ABB RobotStudio station: Solution38RISA.rspag

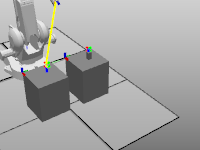
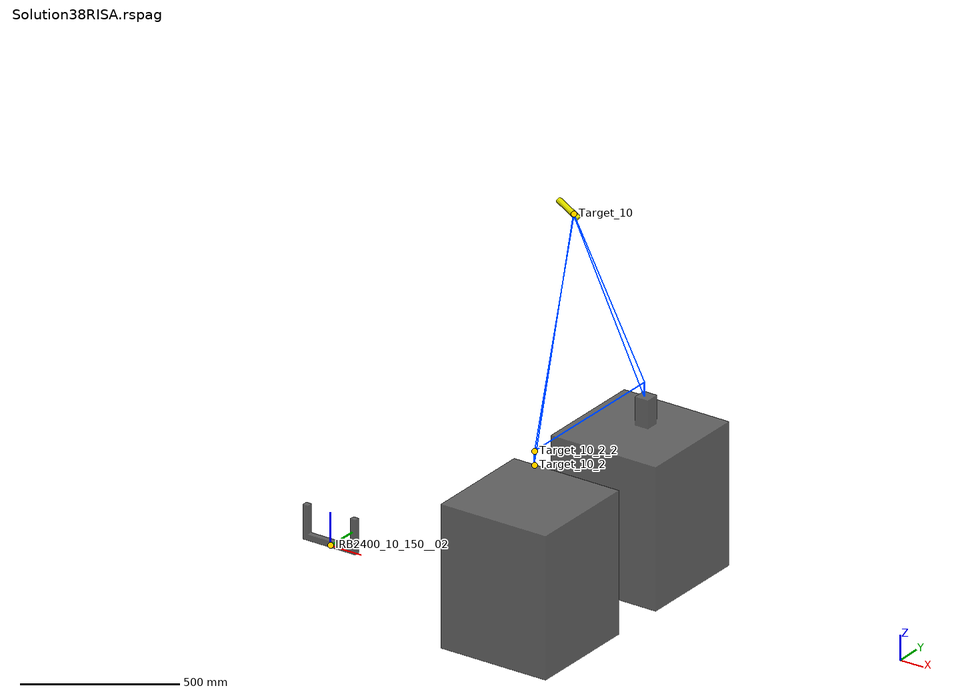
[picture v1: parts stored in the station drawn from their meshes, with robot base, taught points and paths (robot models come from the ABB library and are not in the file)]
--- station ---
Station Solution38RISA (saved by RobotStudio 21.4.9700.0)
Controller IRB2400_10_150
  mechanical unit ROB_1: IRB2400_10_150__02, 6 joints, base frame (0, 0, 0) mm
Layout (positions relative to the parent item):
  - IRB2400_10_150__02 [mechanism, from Robots\IRB2400_10_150_G_02.rslib] at (0, 0, 0) mm; joint values [0, -0.1065, -0.072, 0, 0.5956, 0] (rad or m)
  - Part_4 [part], size 400 x 400 x 500 mm
  - Part_5 [part] at (0, 600, 0) mm, size 400 x 400 x 500 mm
  - Part_6 [part] at (75.01, 607.78, -200) mm, size 50 x 50 x 100 mm
  - Part_1 [part], size 200 x 20 x 20 mm
    - My_Tool1_1 [frame] at (0, 0, 100) mm
  - Part_2 [part], size 20 x 20 x 100 mm
  - Part_3 [part], size 20 x 20 x 100 mm
  - SCGripper1 [smart component] at (842.01, 0, 1462.5) mm, rotated rx -180 ry 60 rz -180 deg
      signals: DI SCOpen, DI SCClose, DO SCClosed, DO SCOpened, DO SCDetal
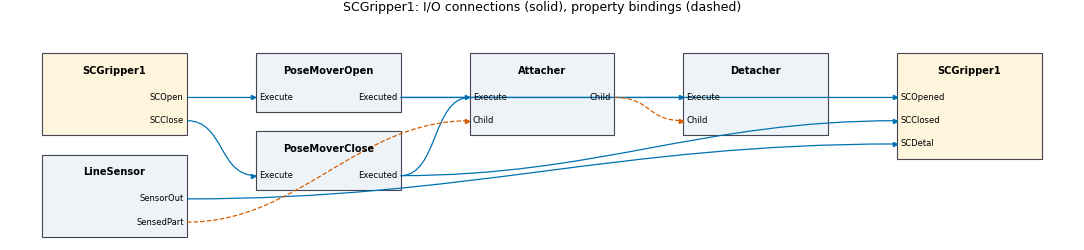
      connections:
        SCGripper1.SCOpen -> PoseMoverOpen.Execute
        SCGripper1.SCClose -> PoseMoverClose.Execute
        PoseMoverOpen.Executed -> SCGripper1.SCOpened
        PoseMoverClose.Executed -> SCGripper1.SCClosed
        LineSensor.SensorOut -> SCGripper1.SCDetal
        PoseMoverClose.Executed -> Attacher.Execute
        PoseMoverOpen.Executed -> Detacher.Execute
        LineSensor.SensedPart => Attacher.Child
        Attacher.Child => Detacher.Child
    - My_Tool1 [mechanism] at (0, 0, 0) mm; joint values [0, 0] (rad or m)
        TCP My_Tool1_1 at (0, 0, 100) mm
        links: L1, L2, L3
    - PoseMoverOpen [smart component, from Components\PoseMover.rslib]
        properties: Mechanism=My_Tool1; Pose=2; Duration=2
    - PoseMoverClose [smart component, from Components\PoseMover.rslib]
        properties: Mechanism=My_Tool1; Pose=3; Duration=2
    - LineSensor [smart component, from Components\LineSensor.rslib]
        properties: Start=[0 0 0.03]; End=[0 0 0.12]; Radius=0.01; SensedPart=(none); SensedPoint=[0 0 0]
      - _sensorPart_ [part], size 20 x 20 x 90 mm
    - Attacher [smart component, from Components\Attacher.rslib]
        properties: Parent=My_Tool1; Flange=0; Child=(none); Mount=false; Offset=[0 0 0]; Orientation=[0 0 0]
    - Detacher [smart component, from Components\Detacher.rslib]
        properties: Child=(none); KeepPosition=true
Attachment: SCGripper1 is attached to IRB2400_10_150__02 / Link6
Attachment: Workobject_1 is attached to Part_4
Attachment: Workobject_2 is attached to Part_5
Collision set CollisionSet_1: My_Tool1 against Part_6, near miss 0 m
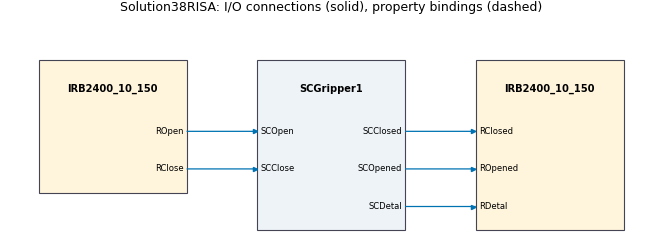
Station logic (signal -> signal, property => property):
  IRB2400_10_150.ROpen -> SCGripper1.SCOpen
  IRB2400_10_150.RClose -> SCGripper1.SCClose
  SCGripper1.SCClosed -> IRB2400_10_150.RClosed
  SCGripper1.SCOpened -> IRB2400_10_150.ROpened
  SCGripper1.SCDetal -> IRB2400_10_150.RDetal
Targets, tools, work objects and paths stored in the station and not in the controller backup, written as RAPID:
! task T_ROB1
MODULE Module1
  CONST robtarget Target_10_2_3:=[[200,225,100],[0,0,1,0],[-1,0,-1,0],[9E+09,9E+09,9E+09,9E+09,9E+09,9E+09]];
  CONST robtarget Target_10_2_2_2:=[[200,225,150],[0,0,1,0],[-1,0,1,0],[9E+09,9E+09,9E+09,9E+09,9E+09,9E+09]];
ENDMODULE


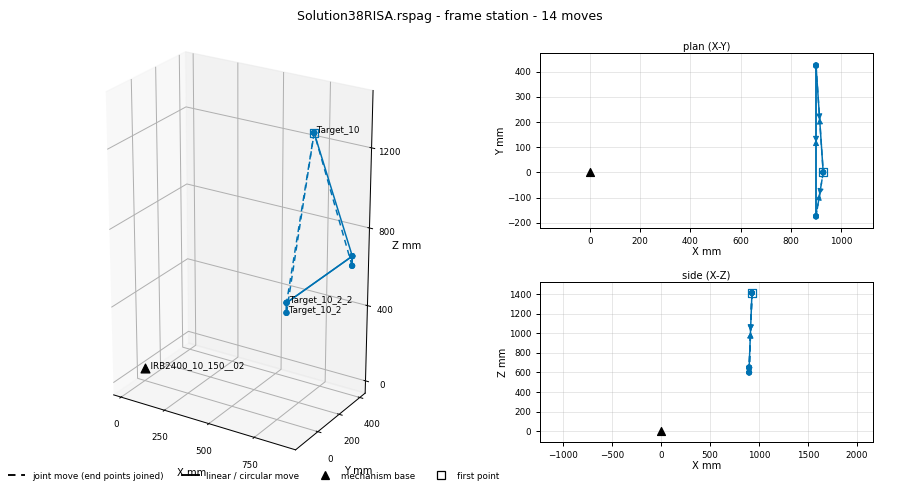
[picture p0: tool path of Solution38RISA.rspag in frame station, 14 of 14 moves have a stored position in this frame; points joined in program order, loops and branches not executed]
--- Backups/IRB2400_10_150/RAPID/TASK1/PROGMOD/CalibData.mod ---
MODULE CalibData
    TASK PERS wobjdata Workobject_1:=[FALSE,TRUE,"",[[700,-400,500],[1,0,0,0]],[[0,0,0],[1,0,0,0]]];
    TASK PERS wobjdata Workobject_2:=[FALSE,TRUE,"",[[700,200,500],[1,0,0,0]],[[0,0,0],[1,0,0,0]]];
    PERS tooldata Tooldata_1:=[TRUE,[[0,0,100],[1,0,0,0]],[1,[0,0,1],[1,0,0,0],0,0,0]];
ENDMODULE

--- Backups/IRB2400_10_150/RAPID/TASK1/PROGMOD/Module1.mod ---
MODULE Module1
        CONST robtarget Target_10:=[[928.612159322,0,1412.5],[0.5,0,0.866025404,0],[0,0,0,0],[9E+09,9E+09,9E+09,9E+09,9E+09,9E+09]];
    CONST robtarget Target_10_2_2:=[[200,225,150],[0,0,1,0],[-1,0,1,0],[9E+09,9E+09,9E+09,9E+09,9E+09,9E+09]];
    CONST robtarget Target_10_2:=[[200,225,100],[0,0,1,0],[-1,0,-1,0],[9E+09,9E+09,9E+09,9E+09,9E+09,9E+09]];
!***********************************************************
    !
    ! Module:  Module1
    !
    ! Description:
    !   <Insert description here>
    !
    ! Author: srk
    !
    ! Version: 1.0
    !
    !***********************************************************


    !***********************************************************
    !
    ! Procedure main
    !
    !   This is the entry point of your program
    !
    !***********************************************************
    PROC main()
        !Add your code here
    ENDPROC
    PROC Path_10()
        MoveJ Target_10,v1000,fine,Tooldata_1\WObj:=wobj0;
        Reset ROpen;
        Reset RClose;
        Set ROpen;
        WaitDI ROpened, 1;
        Reset ROpen;
        MoveJ Target_10_2_2,v1000,z30,Tooldata_1\WObj:=Workobject_1;
        MoveL Target_10_2,v100,fine,Tooldata_1\WObj:=Workobject_1;
        IF RDetal=1 THEN
        Set RClose;
        WaitDI RClosed, 1;
        Reset RClose;
        MoveL Target_10_2_2,v100,z30,Tooldata_1\WObj:=Workobject_1;
        MoveL Target_10_2_2,v1000,z30,Tooldata_1\WObj:=Workobject_2;
        MoveL Target_10_2,v100,fine,Tooldata_1\WObj:=Workobject_2;
        Set ROpen;
        WaitDI ROpened, 1;
        Reset ROpen;
        MoveJ Target_10,v1000,fine,Tooldata_1\WObj:=wobj0;
        EXIT;
        ELSE
            MoveJ Target_10,v1000,fine,Tooldata_1\WObj:=wobj0;
             Reset ROpen;
            Reset RClose;
            Set ROpen;
            WaitDI ROpened, 1;
            Reset ROpen;
            MoveL Target_10_2_2,v1000,z30,Tooldata_1\WObj:=Workobject_2;
            MoveL Target_10_2,v100,fine,Tooldata_1\WObj:=Workobject_2;
            IF RDetal=1 THEN
            Set RClose;
            WaitDI RClosed, 1;
            Reset RClose;
            MoveL Target_10_2_2,v100,z30,Tooldata_1\WObj:=Workobject_2;
            MoveL Target_10_2_2,v1000,z30,Tooldata_1\WObj:=Workobject_1;
            MoveL Target_10_2,v100,fine,Tooldata_1\WObj:=Workobject_1;
            Set ROpen;
            WaitDI ROpened, 1;
            Reset ROpen;

            ENDIF
        ENDIF
        MoveJ Target_10,v1000,fine,Tooldata_1\WObj:=wobj0;


    ENDPROC
ENDMODULE

--- Backups/IRB2400_10_150/SYSPAR/EIO.cfg ---
EIO:CFG_1.0:6:1::
#
EIO_SIGNAL:

      -Name "ROpen" -SignalType "DO" -Label "1"

      -Name "RClose" -SignalType "DO" -Label "2"

      -Name "ROpened" -SignalType "DI" -Label "3"

      -Name "RClosed" -SignalType "DI" -Label "4"

      -Name "RDetal" -SignalType "DI" -Label "5"
